TYPE ST_InputsSection EXTENDS ST_SectionBase :
STRUCT
	nBinInputs		: UINT;
	nIntInputs		: UINT;
	nFloatInputs	: UINT;	
END_STRUCT
END_TYPE

(* stored: Version 1.1.0.1, ProductVersion 3.1.4024.12
   DUT ST_InputsSection: Id {741a8f98-8af3-441d-a86d-fd2ee642c7b4} *)
